(* PLC project Unnamed, Unknown Unnamed 1 *)
(* stored: creationDateTime 2025-12-09T20:40:42, modificationDateTime 2025-12-09T21:00:33 *)

(* Quick little test *)
PROGRAM BasicMirror

            // Quick little test
PROGRAM BasicMirror
VAR
        Input1 AT %IX0.0 : BOOL; // Digital Input (simulatable via debug)
        Output1 AT %QX0.0 : BOOL; // Digital Output
END_VAR

Output1 := Input1; // Boolean mirror assignment, executed per scan cycle

END_PROGRAM
          
END_PROGRAM

CONFIGURATION Config0
  RESOURCE Res0 ON PLC
    TASK task0(INTERVAL := T#20ms, PRIORITY := 0);
    PROGRAM instance0 WITH task0 : BasicMirror;
  END_RESOURCE
END_CONFIGURATION
